// Mitsubishi GX Works2 project: demo-timmer-v2   PLC: FX3U/FX3UC

PROGRAM MAIN
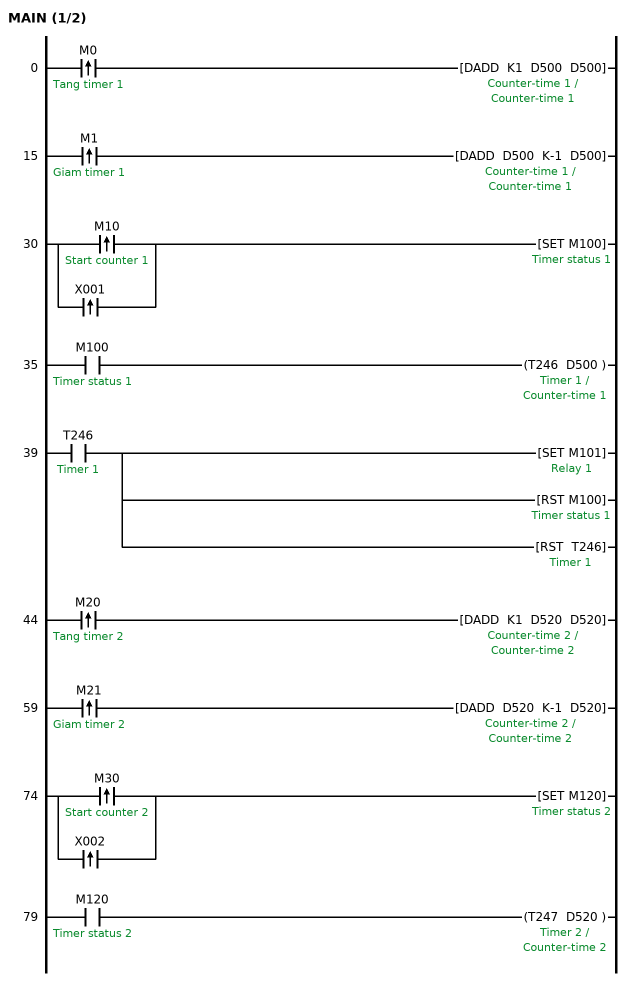
0     LDP     M0  ; Tang timer 1
      DADD    K1 D500 D500  ; Counter-time 1
15    LDP     M1  ; Giam timer 1
      DADD    D500 K-1 D500
30    LDP     M10  ; Start counter 1
      ORP     X001
      SET     M100  ; Timer status 1
35    LD      M100  ; Timer status 1
      OUT     T246 D500  ; Timer 1 / Counter-time 1
39    LD      T246  ; Timer 1
      SET     M101  ; Relay 1
      RST     M100  ; Timer status 1
      RST     T246  ; Timer 1
44    LDP     M20  ; Tang timer 2
      DADD    K1 D520 D520  ; Counter-time 2
59    LDP     M21  ; Giam timer 2
      DADD    D520 K-1 D520
74    LDP     M30  ; Start counter 2
      ORP     X002
      SET     M120  ; Timer status 2
79    LD      M120  ; Timer status 2
      OUT     T247 D520  ; Timer 2 / Counter-time 2
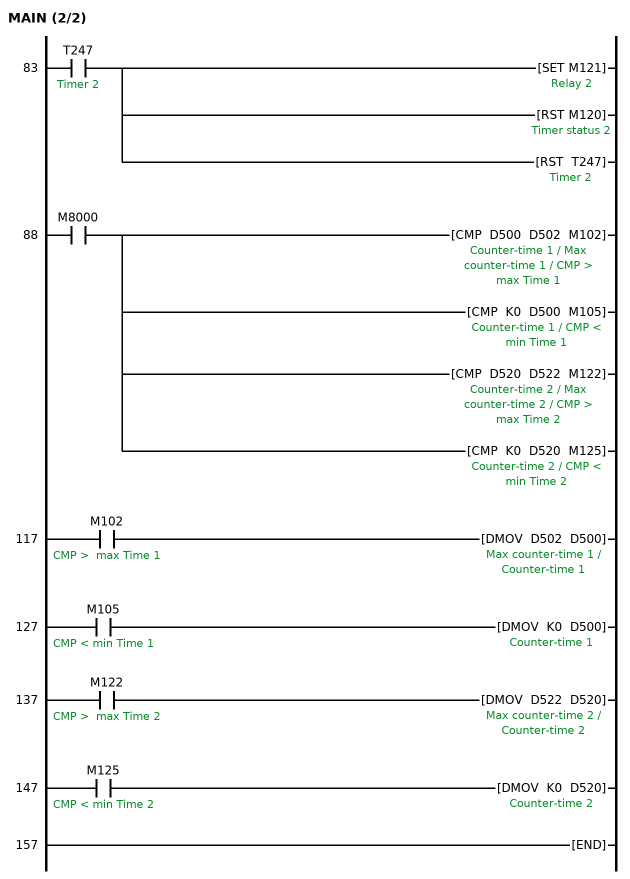
83    LD      T247  ; Timer 2
      SET     M121  ; Relay 2
      RST     M120  ; Timer status 2
      RST     T247  ; Timer 2
88    LD      M8000
      CMP     D500 D502 M102  ; Max counter-time 1 / CMP >  max Time 1
      CMP     K0 D500 M105  ; CMP < min Time 1
      CMP     D520 D522 M122  ; Max counter-time 2 / CMP >  max Time 2
      CMP     K0 D520 M125  ; CMP < min Time 2
117   LD      M102  ; CMP >  max Time 1
      DMOV    D502 D500
127   LD      M105  ; CMP < min Time 1
      DMOV    K0 D500
137   LD      M122  ; CMP >  max Time 2
      DMOV    D522 D520
147   LD      M125  ; CMP < min Time 2
      DMOV    K0 D520
157   END
END_PROGRAM

// device comments not shown above
M103  ; CMP = max Time 1
M104  ; CMP <  max Time 1
M106  ; CMP =  min Time 1
M107  ; CMP >  min Time 1
M123  ; CMP = max Time 2
M124  ; CMP <  max Time 2
M126  ; CMP =  min Time 2
M127  ; CMP >  min Time
T426  ; Timer 1
